// TIA Portal V16 export
// export: Created 2025-12-18T09:29:14.9442788Z, ExportSetting WithDefaults, DisplayName Totally Integrated Automation Portal, DisplayVersion V16, DisplayName TIA Portal Version Control Interface, DisplayVersion V16, DisplayName TIA Portal Openness, DisplayVersion V16, DisplayName STEP 7 Professional, DisplayVersion V16, DisplayName STEP 7 Safety, DisplayVersion V16, DisplayName WinCC Advanced, DisplayVersion V16
FUNCTION_BLOCK "Control Panel"   // FB2, LAD
{ S7_Optimized_Access := 'TRUE' }
VERSION : 0.1
// stored: AutoNumber true, IsIECCheckEnabled false, IsRetainMemResEnabled false, MemoryReserve 100, SetENOAutomatically false, UDAEnableTagReadback false
   VAR_INPUT
      xResetButton : Bool;
      xEmergencyButton : Bool;
   END_VAR
   VAR_IN_OUT
      xProcessLight : Bool;
      diProcessTimeLeft : DInt;
      "Work Station DB" : "UDT WorkStation";
   END_VAR
   VAR
      diProcessTime : DInt;
   END_VAR
BEGIN

REGION Network 1
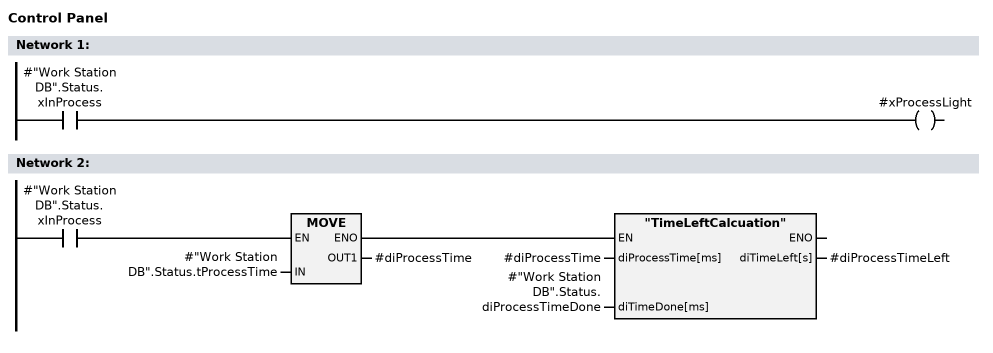
   RUNG wire#powerrail
      Contact( #"Work Station DB".Status.xInProcess )
      Coil( #xProcessLight )
   END_RUNG
   // the same network as SCL:
   #xProcessLight := #"Work Station DB".Status.xInProcess;
END_REGION

REGION Network 2
   RUNG wire#powerrail
      Contact( #"Work Station DB".Status.xInProcess )
      Move(in := #"Work Station DB".Status.tProcessTime, out1 => #diProcessTime)
      "TimeLeftCalcuation"("diProcessTime[ms]" := #diProcessTime, "diTimeDone[ms]" := #"Work Station DB".Status.diProcessTimeDone, "diTimeLeft[s]" => #diProcessTimeLeft)
   END_RUNG
   // the same network as SCL:
   IF #"Work Station DB".Status.xInProcess THEN
       #diProcessTime := #"Work Station DB".Status.tProcessTime;
       "TimeLeftCalcuation"("diProcessTime[ms]" := #diProcessTime,
                            "diTimeDone[ms]" := #"Work Station DB".Status.diProcessTimeDone,
                            "diTimeLeft[s]" => #diProcessTimeLeft);
   END_IF;
END_REGION
END_FUNCTION_BLOCK
